FUNCTION TryConvert_TOD_TO_BYTE : BOOL
VAR_INPUT
	in : TOD;
	out : REFERENCE TO BYTE;
END_VAR

IF in > DatatypeLimits.MAX_VALUE_OF_TOD_WHICH_CAN_BE_HELD_IN_A_BYTE THEN
	RETURN;
END_IF

out := TOD_TO_BYTE(in);
TryConvert_TOD_TO_BYTE := TRUE;

END_FUNCTION

(* stored: Version 1.1.0.1, ProductVersion 3.1.4024.12
   POU TryConvert_TOD_TO_BYTE: Id {a3200b40-eeac-4dd1-b775-adc4a7142fd7}, SpecialFunc None *)
